FUNCTION_BLOCK "CPG_RecipeSetpoint_BOOL"
TITLE = CPG_RecipeSetpoint_BOOL
{ S7_Optimized_Access := 'TRUE' }
AUTHOR : 'tech.team.motioncontrol@siemens.com'
FAMILY : CPG
VERSION : 1.1
//Support: tech.team.motioncontrol@siemens.com
   VAR_INPUT
      enable { ExternalAccessible := 'False'; ExternalVisible := 'False'; ExternalWritable := 'False'} : Bool;   // If true, setpoint changes are permitted
      disableRecipeControl { ExternalAccessible := 'False'; ExternalVisible := 'False'; ExternalWritable := 'False'} : Bool;   // If true, the setpoint is no longer handled as a recipe
   END_VAR

   VAR_OUTPUT
      out { ExternalAccessible := 'False'; ExternalVisible := 'False'; ExternalWritable := 'False'} : Bool;   // Currently running recipe value
      changeEnabled { ExternalAccessible := 'False'; ExternalVisible := 'False'; ExternalWritable := 'False'} : Bool;   // Enable input is true, setpoint can be changed
      recipeControlDisabled { ExternalAccessible := 'False'; ExternalVisible := 'False'; ExternalWritable := 'False'} : Bool;   // The value is not subject to recipe controls
      changeNotAllowed { ExternalAccessible := 'False'; ExternalVisible := 'False'; ExternalWritable := 'False'} : Bool;   // Change is not permitted due to machine state
      recipeSetpointDifference { ExternalAccessible := 'False'; ExternalVisible := 'False'; ExternalWritable := 'False'} : Bool;   // The currently running (out) value and setpoint value are not equal
   END_VAR

   VAR_IN_OUT
      recipeControl : "CPG_typeRecipeControl";   // Recipe control tag
      recipeSetpoint : "CPG_typeRecipeSetpoint_BOOL";   // Recipe setpoint tag
   END_VAR

   VAR
      statFirstScan { ExternalAccessible := 'False'; ExternalVisible := 'False'; ExternalWritable := 'False'} : Bool := true;
      statPrevChangeNum { ExternalAccessible := 'False'; ExternalVisible := 'False'; ExternalWritable := 'False'} : Int;
      statPrevSaveNum { ExternalAccessible := 'False'; ExternalVisible := 'False'; ExternalWritable := 'False'} : Int;
      statPrevCopyNum { ExternalAccessible := 'False'; ExternalVisible := 'False'; ExternalWritable := 'False'} : Int;
      statPrevDeleteNum { ExternalAccessible := 'False'; ExternalVisible := 'False'; ExternalWritable := 'False'} : Int;
      statPrevOut { ExternalAccessible := 'False'; ExternalVisible := 'False'; ExternalWritable := 'False'} : Bool;
      statChangeNotAllowedTimer {InstructionName := 'TON_TIME'; LibVersion := '1.0'; ExternalAccessible := 'False'; ExternalVisible := 'False'; ExternalWritable := 'False'} : TON_TIME;
      statTimerEN { ExternalAccessible := 'False'; ExternalVisible := 'False'; ExternalWritable := 'False'} : Bool;
   END_VAR

   VAR CONSTANT
      DELAY_TIME : Time := T#3s;
   END_VAR


BEGIN
	//============================================================================================================
	// SIEMENS AG
	// (c)Copyright 2019 All Rights Reserved
	//------------------------------------------------------------------------------------------------------------
	// Library: LCPG
	// Tested with: S7-1500 with FW version V2.1
	// Engineering: TIA Portal V14
	// Restrictions: ---
	// Requirements: S7-1500
	// Functionality: instantiate this once in the program for each recipe setpoint of BOOL
	// Support: tech.team.motioncontrol@siemens.com
	//------------------------------------------------------------------------------------------------------------
	// Change log table:
	// Version       Date               Expert in charge    Changes applied
	//  01.01.00     02.01.2019         KB                  Initial Release
	//============================================================================================================
	// Function : CPG_RecipeSetpoint_BOOL
	//============================================================================================================

	// Language Selection
	#recipeSetpoint.CurrentName := #recipeSetpoint.SetpointName[#recipeControl.LanguageSelection];
	#recipeSetpoint.CurrentTextFalse := #recipeSetpoint.Text_False[#recipeControl.LanguageSelection];
	#recipeSetpoint.CurrentTextTrue := #recipeSetpoint.Text_True[#recipeControl.LanguageSelection];

	//Recipe Disable Control
	#recipeSetpoint.DisableRecipeControl := #disableRecipeControl;

	//Pass through enable bit
	#recipeSetpoint.SetpointChangeEnabled := #enable;

	//Set out value to match initial one on first scan
	IF #statFirstScan THEN
	    #recipeSetpoint.CurrentRecipeValue := #recipeSetpoint.RecipeValues[#recipeControl.CurrentRecipeID];
	    #recipeSetpoint.OUT := #recipeSetpoint.RecipeValues[#recipeControl.CurrentRecipeID];
	    #statFirstScan := false;
	END_IF;


	REGION RECIPE CONTROL
	    // Recipe Control - Change, Save, Copy, Delete, Revert setpoint, Save setpoint
	    IF NOT (#recipeSetpoint.DisableRecipeControl) THEN
	        //Recipe Change Command
	        IF #recipeControl.RecipeChangeNum <> #statPrevChangeNum THEN
	            #recipeSetpoint.OUT := #recipeSetpoint.RecipeValues[#recipeControl.CurrentRecipeID];
	            #statPrevChangeNum := #recipeControl.RecipeChangeNum;
	            // Prevents multiple commands from being executed if this instruction is not being scanned
	            #statPrevSaveNum := #recipeControl.RecipeSaveNum;
	            #statPrevCopyNum := #recipeControl.RecipeCopyNum;
	            #statPrevDeleteNum := #recipeControl.RecipeDeleteNum;
	        END_IF;
	        //Recipe Save Command
	        IF #recipeControl.RecipeSaveNum <> #statPrevSaveNum THEN
	            #recipeSetpoint.RecipeValues[#recipeControl.RecipeDestinationID] := #recipeSetpoint.OUT;
	            #statPrevSaveNum := #recipeControl.RecipeSaveNum;
	            // Prevents multiple commands from being executed if this instruction is not being scanned
	            #statPrevCopyNum := #recipeControl.RecipeCopyNum;
	            #statPrevDeleteNum := #recipeControl.RecipeDeleteNum;
	        END_IF;
	        //Recipe Copy Command
	        IF #recipeControl.RecipeCopyNum <> #statPrevCopyNum THEN
	            #recipeSetpoint.RecipeValues[#recipeControl.RecipeDestinationID] := #recipeSetpoint.RecipeValues[#recipeControl.RecipeSourceID];
	            #statPrevCopyNum := #recipeControl.RecipeCopyNum;
	            // Prevents multiple commands from being executed if this instruction is not being scanned
	            #statPrevDeleteNum := #recipeControl.RecipeDeleteNum;
	        END_IF;
	        //Recipe Delete Command
	        IF #recipeControl.RecipeDeleteNum <> #statPrevDeleteNum THEN
	            //edit this line to change the value a deleted recipe defaults to
	            #recipeSetpoint.RecipeValues[#recipeControl.RecipeDestinationID] := false;
	            #statPrevDeleteNum := #recipeControl.RecipeDeleteNum;
	        END_IF;
	        // Revert setpoint to saved value
	        IF #recipeSetpoint.RevertSetpoint THEN
	            #recipeSetpoint.OUT := #recipeSetpoint.RecipeValues[#recipeControl.CurrentRecipeID];
	        END_IF;
	        //Detect recipe/setpoint difference
	        IF (#recipeSetpoint.RecipeValues[#recipeControl.CurrentRecipeID] <> #recipeSetpoint.OUT) AND NOT (#recipeControl.RecipeChange) THEN
	            #recipeControl.RecipeSetpointDiff := true;  //signal to recipe control that a setpoint differs
	            #recipeSetpoint.RecipeSetpointDiff := true;
	        ELSE
	            #recipeSetpoint.RecipeSetpointDiff := false;
	        END_IF;
	        //Save setpoint
	        IF #recipeSetpoint.SaveSetpoint THEN
	            #recipeSetpoint.RecipeValues[#recipeControl.CurrentRecipeID] := #recipeSetpoint.OUT;
	        END_IF;

	        //update values stored for current recipe & recipes A, B, & C
	        #recipeSetpoint.CurrentRecipeValue := #recipeSetpoint.RecipeValues[#recipeControl.CurrentRecipeID];
	        #recipeSetpoint.RecipeValueA := #recipeSetpoint.RecipeValues[#recipeControl.RecipeID_A];
	        #recipeSetpoint.RecipeValueB := #recipeSetpoint.RecipeValues[#recipeControl.RecipeID_B];
	        #recipeSetpoint.RecipeValueC := #recipeSetpoint.RecipeValues[#recipeControl.RecipeID_C];

	    ELSE    //if recipe control is disabled, just update counters
	        #recipeSetpoint.RecipeSetpointDiff := false;
	        #statPrevChangeNum := #recipeControl.RecipeChangeNum;
	        #statPrevSaveNum := #recipeControl.RecipeSaveNum;
	        #statPrevCopyNum := #recipeControl.RecipeCopyNum;
	        #statPrevDeleteNum := #recipeControl.RecipeDeleteNum;
	    END_IF;
	END_REGION


	REGION UPDATE IN VALUE
	    //If ENABLE, then changes to the setpoint value are possible
	    //otherwise, updating the setpoint is not possible via changing RecipeSetpoint.IN
	    IF #enable THEN
	        //Clear status bit
	        #recipeSetpoint.SetpointChangeDisabled := false;

	        // Check for input changed (due to user updating RecipeSetpoint.IN)
	        IF (#recipeSetpoint.IN XOR #recipeSetpoint.OUT) AND NOT (#recipeSetpoint.OUT XOR #statPrevOut) THEN
	            #recipeSetpoint.OUT := #recipeSetpoint.IN;
	        ELSE  // otherwise, update in to match out (this branch can execute due to a recipe change)
	            #recipeSetpoint.IN := #recipeSetpoint.OUT;
	        END_IF;

	    ELSE

	        // If in changes, revert and display message
	        IF (#recipeSetpoint.IN XOR #recipeSetpoint.OUT) OR #recipeSetpoint.RevertSetpoint THEN
	            #recipeSetpoint.IN := #recipeSetpoint.OUT;
	            #statTimerEN := false;
	            #recipeSetpoint.SetpointChangeDisabled := true;
	        END_IF;

	        //display "setpoint changes not allowed" 3 seconds after inputting an invalid change
	        #statChangeNotAllowedTimer(IN := #statTimerEN,
	                               PT := #DELAY_TIME);

	        // Continue to display the status bits for the duration of the timer.
	        IF #recipeSetpoint.SetpointChangeDisabled THEN
	            #statTimerEN := true;
	            #recipeSetpoint.SetpointChangeDisabled :=
	                #recipeSetpoint.SetpointChangeDisabled AND #statTimerEN AND NOT #statChangeNotAllowedTimer.Q;
	        END_IF;

	    END_IF;
	END_REGION


	REGION DETERMINE HMI TEXTS
	    //This is a workaround because multiplexing inside a faceplate is not possible in V14SP1
	    IF #recipeSetpoint.OUT THEN
	        #recipeSetpoint.Out_Text := #recipeSetpoint.CurrentTextTrue;
	    ELSE
	        #recipeSetpoint.Out_Text := #recipeSetpoint.CurrentTextFalse;
	    END_IF;
	    IF #recipeSetpoint.CurrentRecipeValue THEN
	        #recipeSetpoint.CurrentRecipeValue_Text := #recipeSetpoint.CurrentTextTrue;
	    ELSE
	        #recipeSetpoint.CurrentRecipeValue_Text := #recipeSetpoint.CurrentTextFalse;
	    END_IF;
	    IF #recipeSetpoint.RecipeValueA THEN
	        #recipeSetpoint.RecipeA_Text := #recipeSetpoint.CurrentTextTrue;
	    ELSE
	        #recipeSetpoint.RecipeA_Text := #recipeSetpoint.CurrentTextFalse;
	    END_IF;
	    IF #recipeSetpoint.RecipeValueB THEN
	        #recipeSetpoint.RecipeB_Text := #recipeSetpoint.CurrentTextTrue;
	    ELSE
	        #recipeSetpoint.RecipeB_Text := #recipeSetpoint.CurrentTextFalse;
	    END_IF;
	    IF #recipeSetpoint.RecipeValueC THEN
	        #recipeSetpoint.RecipeC_Text := #recipeSetpoint.CurrentTextTrue;
	    ELSE
	        #recipeSetpoint.RecipeC_Text := #recipeSetpoint.CurrentTextFalse;
	    END_IF;
	END_REGION


	REGION SET OUTPUTS
	    #out := #recipeSetpoint.OUT;
	    #statPrevOut := #recipeSetpoint.OUT;
	    #changeNotAllowed := #recipeSetpoint.SetpointChangeDisabled;
	    #recipeSetpointDifference := #recipeSetpoint.RecipeSetpointDiff;
	    #recipeControlDisabled := #recipeSetpoint.DisableRecipeControl;
	    #changeEnabled := #recipeSetpoint.SetpointChangeEnabled;
	END_REGION


	//  -------------- END OF LOGIC -------------------------
	ENO := TRUE;   // Set the ENO output
END_FUNCTION_BLOCK

